Omron Sysmac Studio project Cobot Modbus Test_100221 (Sysmac Studio 1.40.0.64008, StandardProject)

# Controller new_Controller_0: NX102-9020 version 1.34
Units and slaves: Unit 1 : NX-OC4633 (N1)
Task PrimaryTask (priority 4, period or condition 2000): Main, TM_Movements_Connection, TM_Movements, CobotModbusComms
Library TM_Commands 1.2.1 (contents left out)
Library TMmodbus Lib FW1.80 FB3.0.03 3.0.03 (contents left out)

VAR_GLOBAL RETAIN
    StartCommunications : BOOL;  (* published *)
END_VAR
VAR_GLOBAL
    MBerror : WORD;  (* published *)
    RobotCoordinates : TMmodbus\sRobotCoordinate;  (* published *)
    TouchCoordinates : TMmodbus\sRobotCoordinateTouch;  (* published *)
    RobotStatus : TMmodbus\sRobotStatus;  (* published *)
    RobotVitals : TMmodbus\sRobotVitals;  (* published *)
    Config : TMmodbus\sConfiguration;  (* published *)
    RobotJointTorques : TMmodbus\sRobotJointTorque;  (* published *)
    RobotTCPLive : TMmodbus\sRobotTCPLive;  (* published *)
    CurrentProjectName : string[200];  (* published *)
    NewProjectName : string[200];  (* published *)
    CommsRoundRobin : REAL;  (* published *)
    TCPerror : WORD;  (* published *)
    RobotControlBoxInfo : TMmodbus\sRobotControllerData;  (* published *)
    Buttons : TMmodbus\sRobotStickButtons;  (* published *)
    RobotIO : TMmodbus\sRobotIO;  (* published *)
    RobotSafetySettings : TMmodbus\sRobotSafety;  (* published *)
    RealsToRobot : ARRAY[0..49] OF real;  (* published *)
    FloatsFromRobot : ARRAY[0..49] OF real;  (* published *)
    BoolsToRobot : ARRAY[0..63] OF BOOL;  (* published *)
    Int16sFromRobot : ARRAY[0..49] OF INT;  (* published *)
    BoolsFromRobot : ARRAY[0..63] OF BOOL;  (* published *)
    IntsToRobot : ARRAY[0..49] OF INT;  (* published *)
    CommunicationsStatus : _eCONNECTION_STATE;  (* published *)
    CommunicationsBusy : BOOL;  (* published *)
    TCPerrorOriginator : TMModbus\eFunctionBlockError;  (* published *)
    RetryCounter : UINT;  (* published *)
    Stitching_Status : DINT;  (* published *)
    Stitching_Speed : REAL;  (* published *)
    Robot_Status : DINT;  (* published *)
    RobPos_X : REAL;  (* published *)
    RobPos_Y : REAL;  (* published *)
    RobPos_Z : REAL;  (* published *)
    Relay_Output : BYTE;  (* at IOBus://unit#1/Output Bit 8 bits; published *)
    Relay_Output1 : BOOL;  (* at IOBus://unit#1/Output Bit 8 bits/Output Bit 00; published *)
    Relay_Output2 : BOOL;  (* at IOBus://unit#1/Output Bit 8 bits/Output Bit 01; published *)
    Relay_Output3 : BOOL;  (* at IOBus://unit#1/Output Bit 8 bits/Output Bit 02; published *)
    Relay_Output4 : BOOL;  (* at IOBus://unit#1/Output Bit 8 bits/Output Bit 03; published *)
    Run_Stiching : BOOL;  (* published *)
    StartProgram : BOOL;  (* published *)
    CableConnected : BOOL;  (* published *)
    MTCP_Connect_TCP_Socket : _sSOCKET;  (* published *)
    MTCP_Connect_Connected : BOOL;
    ListenNode_Connect_Connected : BOOL;
    ListenNode_Connect_TCP_Socket : _sSOCKET;
    TaskTimeFB : REAL;
    Speed : REAL;  (* published *)
    TM_ReadPosition_X : REAL;
    TM_ReadPosition_Y : REAL;
    TM_ReadPosition_Z : REAL;  (* published *)
    Register : ARRAY[0..1023] OF WORD;
    TM_MovCmd_Command : STRING[256];
    Stitching_InManual : BOOL;
    Vision_IN : ARRAY[0..495] OF BYTE;  (* network input *)
    Vision_IN_Bit : ARRAY[0..11] OF BYTE;  (* network input *)
    Vision_Out_Bit : ARRAY[0..11] OF BYTE;  (* network output *)
    Vision_OUT : ARRAY[0..495] OF BYTE;  (* network output *)
END_VAR

PROGRAM Main
VAR
    Input1 : BOOL;  (* Enter Variable Commen *)
    Input2 : BOOL;
    Input3 : BOOL;
    Input4 : BOOL;
    RobotPos_Stiching : BOOL;
    xPlaceholder : DINT;
    yPlaceholder : DINT;
    zPlaceholder : DINT;
    placeholder : BOOL;
    Robot_Running : BOOL;
    Rb_Error_Present : BOOL;
    St_Error_Present : BOOL;
    CommunicationsBusy : BOOL;
    StartCommunications : BOOL;
    Start : BOOL;
    test : BOOL;
    def : BOOL;
    Angle : BOOL;
    Part_Orientation : INT;
    Part_Orientation_REAL : REAL;
    Part_Orientation_DINT : DINT;
    Part_Dist_X : DINT;
    Part_Dist_Y : DINT;
END_VAR
VAR_EXTERNAL
    Stitching_Status : DINT;
    Stitching_Speed : REAL;
    Robot_Status : DINT;
    Relay_Output : BYTE;
    RobPos_X : REAL;
    RobPos_Y : REAL;
    RobPos_Z : REAL;
    RobotCoordinates : TMmodbus\sRobotCoordinate;
    RobotStatus : TMmodbus\sRobotStatus;
    Run_Stiching : BOOL;
    Speed : REAL;
    Vision_IN : ARRAY[0..495] OF BYTE;
END_VAR

(* Section DataToGrafana: ladder, written here as Structured Text *)

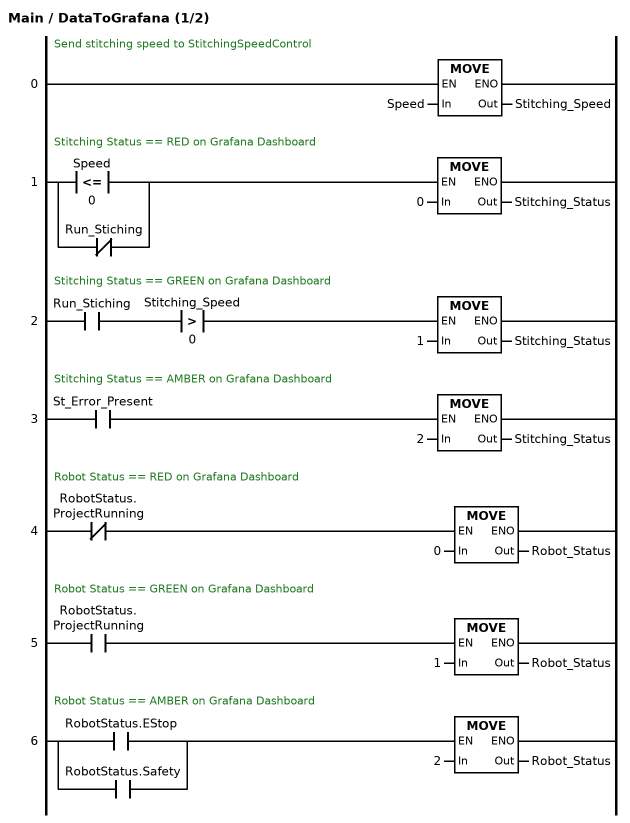
(* Rung 0: Send stitching speed to StitchingSpeedControl *)
Stitching_Speed := Speed;
(* Rung 1: Stitching Status == RED on Grafana Dashboard *)
IF (Speed <= 0) OR NOT Run_Stiching THEN Stitching_Status := 0; END_IF;
(* Rung 2: Stitching Status == GREEN on Grafana Dashboard *)
IF Run_Stiching AND (Stitching_Speed > 0) THEN Stitching_Status := 1; END_IF;
(* Rung 3: Stitching Status == AMBER on Grafana Dashboard *)
IF St_Error_Present THEN Stitching_Status := 2; END_IF;
(* Rung 4: Robot Status == RED on Grafana Dashboard *)
IF NOT RobotStatus.ProjectRunning THEN Robot_Status := 0; END_IF;
(* Rung 5: Robot Status == GREEN on Grafana Dashboard *)
IF RobotStatus.ProjectRunning THEN Robot_Status := 1; END_IF;
(* Rung 6: Robot Status == AMBER on Grafana Dashboard *)
IF RobotStatus.EStop OR RobotStatus.Safety THEN Robot_Status := 2; END_IF;

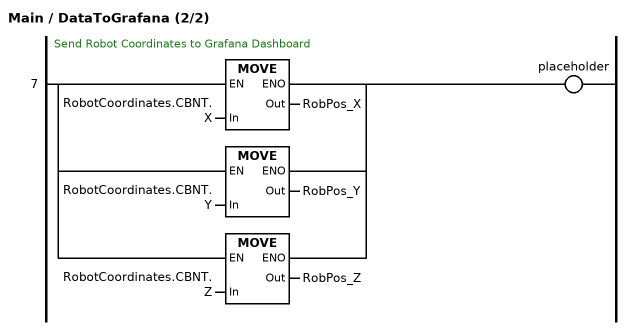
(* Rung 7: Send Robot Coordinates to Grafana Dashboard *)
RobPos_X := RobotCoordinates.CBNT.X;
RobPos_Y := RobotCoordinates.CBNT.Y;
RobPos_Z := RobotCoordinates.CBNT.Z;
placeholder := TRUE;

(* Section StichingSpeedControl: ladder, written here as Structured Text *)

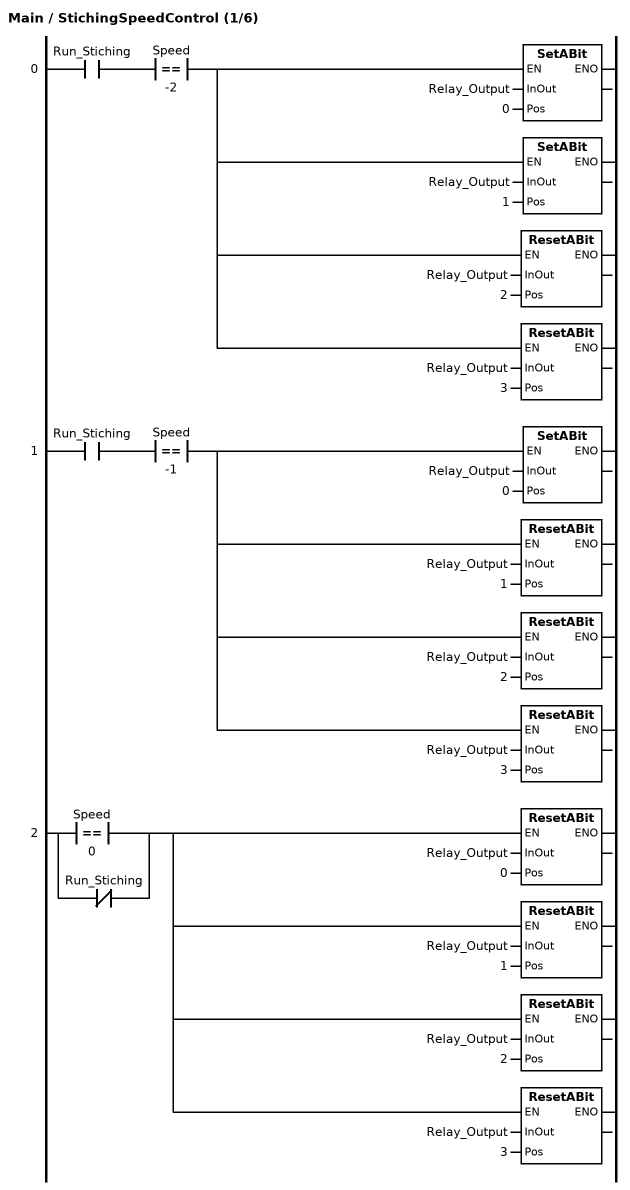
(* Rung 0 *)
IF Run_Stiching AND (Speed = -2) THEN
    SetABit(InOut := Relay_Output, Pos := 0);
    SetABit(InOut := Relay_Output, Pos := 1);
    ResetABit(InOut := Relay_Output, Pos := 2);
    ResetABit(InOut := Relay_Output, Pos := 3);
END_IF;
(* Rung 1 *)
IF Run_Stiching AND (Speed = -1) THEN
    SetABit(InOut := Relay_Output, Pos := 0);
    ResetABit(InOut := Relay_Output, Pos := 1);
    ResetABit(InOut := Relay_Output, Pos := 2);
    ResetABit(InOut := Relay_Output, Pos := 3);
END_IF;
(* Rung 2 *)
IF (Speed = 0) OR NOT Run_Stiching THEN
    ResetABit(InOut := Relay_Output, Pos := 0);
    ResetABit(InOut := Relay_Output, Pos := 1);
    ResetABit(InOut := Relay_Output, Pos := 2);
    ResetABit(InOut := Relay_Output, Pos := 3);
END_IF;

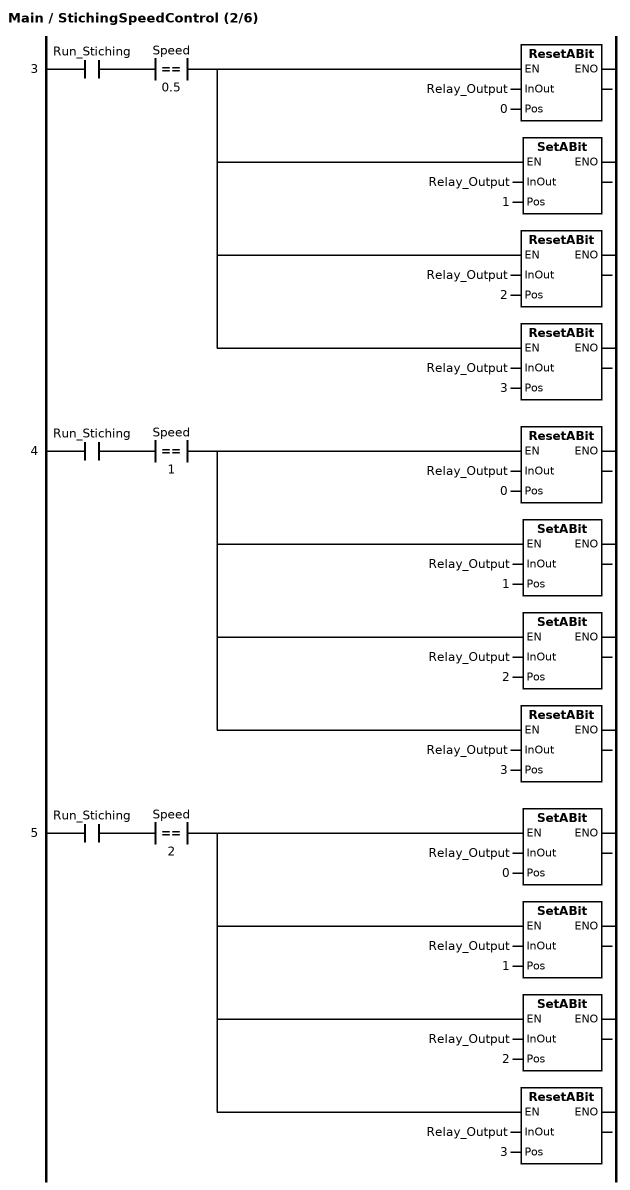
(* Rung 3 *)
IF Run_Stiching AND (Speed = 0.5) THEN
    ResetABit(InOut := Relay_Output, Pos := 0);
    SetABit(InOut := Relay_Output, Pos := 1);
    ResetABit(InOut := Relay_Output, Pos := 2);
    ResetABit(InOut := Relay_Output, Pos := 3);
END_IF;
(* Rung 4 *)
IF Run_Stiching AND (Speed = 1) THEN
    ResetABit(InOut := Relay_Output, Pos := 0);
    SetABit(InOut := Relay_Output, Pos := 1);
    SetABit(InOut := Relay_Output, Pos := 2);
    ResetABit(InOut := Relay_Output, Pos := 3);
END_IF;
(* Rung 5 *)
IF Run_Stiching AND (Speed = 2) THEN
    SetABit(InOut := Relay_Output, Pos := 0);
    SetABit(InOut := Relay_Output, Pos := 1);
    SetABit(InOut := Relay_Output, Pos := 2);
    ResetABit(InOut := Relay_Output, Pos := 3);
END_IF;

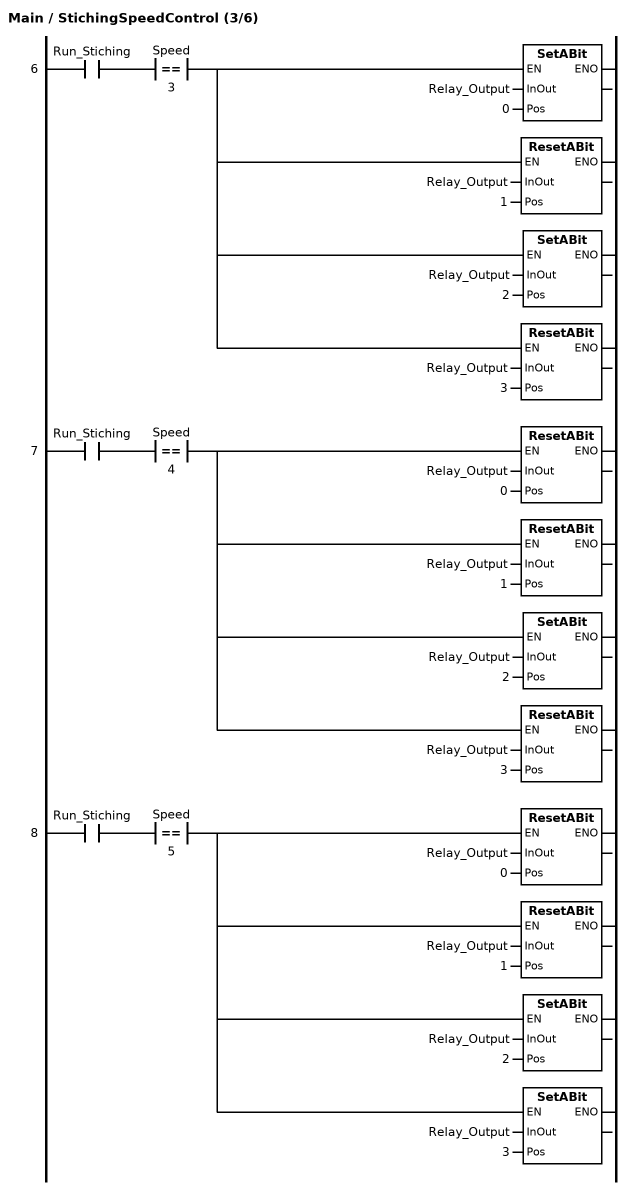
(* Rung 6 *)
IF Run_Stiching AND (Speed = 3) THEN
    SetABit(InOut := Relay_Output, Pos := 0);
    ResetABit(InOut := Relay_Output, Pos := 1);
    SetABit(InOut := Relay_Output, Pos := 2);
    ResetABit(InOut := Relay_Output, Pos := 3);
END_IF;
(* Rung 7 *)
IF Run_Stiching AND (Speed = 4) THEN
    ResetABit(InOut := Relay_Output, Pos := 0);
    ResetABit(InOut := Relay_Output, Pos := 1);
    SetABit(InOut := Relay_Output, Pos := 2);
    ResetABit(InOut := Relay_Output, Pos := 3);
END_IF;
(* Rung 8 *)
IF Run_Stiching AND (Speed = 5) THEN
    ResetABit(InOut := Relay_Output, Pos := 0);
    ResetABit(InOut := Relay_Output, Pos := 1);
    SetABit(InOut := Relay_Output, Pos := 2);
    SetABit(InOut := Relay_Output, Pos := 3);
END_IF;

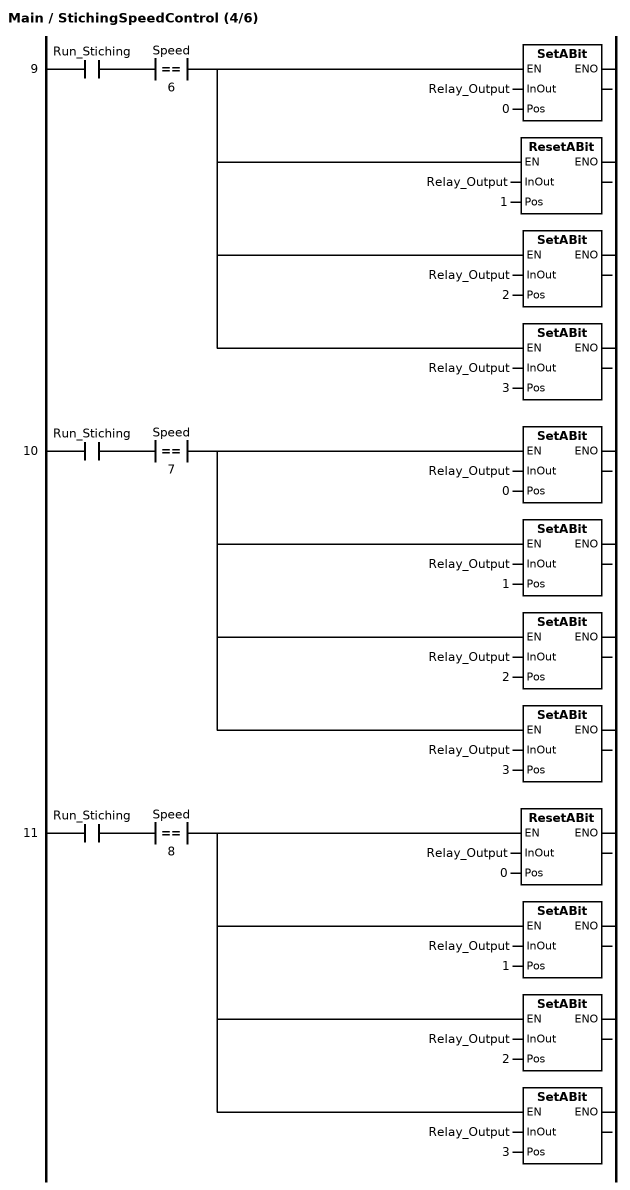
(* Rung 9 *)
IF Run_Stiching AND (Speed = 6) THEN
    SetABit(InOut := Relay_Output, Pos := 0);
    ResetABit(InOut := Relay_Output, Pos := 1);
    SetABit(InOut := Relay_Output, Pos := 2);
    SetABit(InOut := Relay_Output, Pos := 3);
END_IF;
(* Rung 10 *)
IF Run_Stiching AND (Speed = 7) THEN
    SetABit(InOut := Relay_Output, Pos := 0);
    SetABit(InOut := Relay_Output, Pos := 1);
    SetABit(InOut := Relay_Output, Pos := 2);
    SetABit(InOut := Relay_Output, Pos := 3);
END_IF;
(* Rung 11 *)
IF Run_Stiching AND (Speed = 8) THEN
    ResetABit(InOut := Relay_Output, Pos := 0);
    SetABit(InOut := Relay_Output, Pos := 1);
    SetABit(InOut := Relay_Output, Pos := 2);
    SetABit(InOut := Relay_Output, Pos := 3);
END_IF;

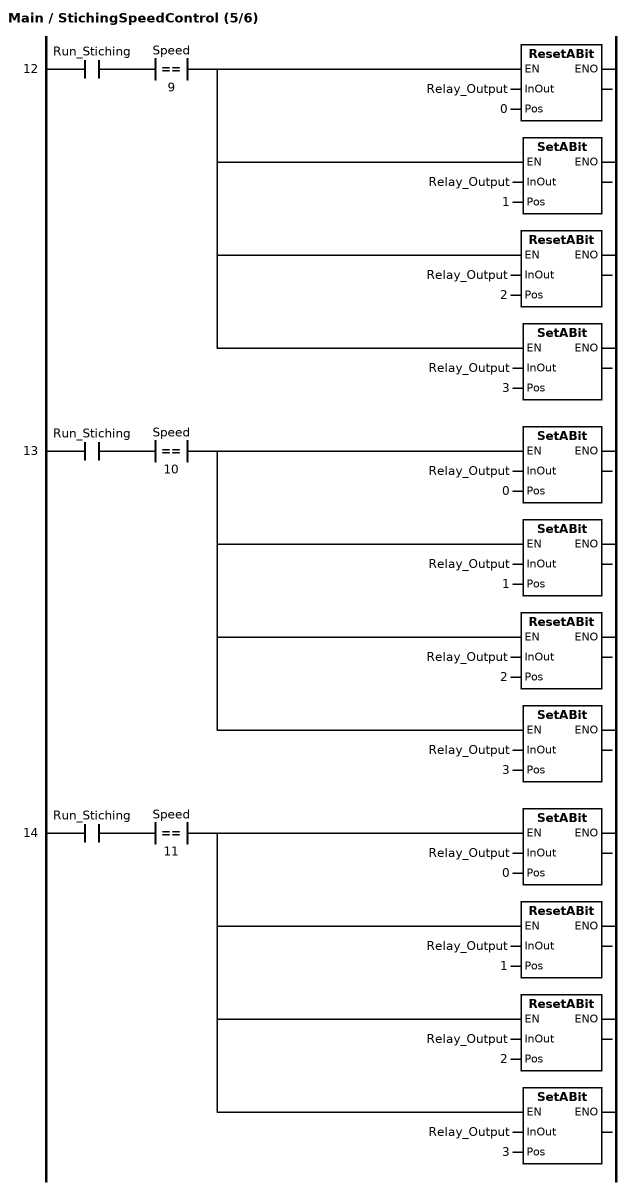
(* Rung 12 *)
IF Run_Stiching AND (Speed = 9) THEN
    ResetABit(InOut := Relay_Output, Pos := 0);
    SetABit(InOut := Relay_Output, Pos := 1);
    ResetABit(InOut := Relay_Output, Pos := 2);
    SetABit(InOut := Relay_Output, Pos := 3);
END_IF;
(* Rung 13 *)
IF Run_Stiching AND (Speed = 10) THEN
    SetABit(InOut := Relay_Output, Pos := 0);
    SetABit(InOut := Relay_Output, Pos := 1);
    ResetABit(InOut := Relay_Output, Pos := 2);
    SetABit(InOut := Relay_Output, Pos := 3);
END_IF;
(* Rung 14 *)
IF Run_Stiching AND (Speed = 11) THEN
    SetABit(InOut := Relay_Output, Pos := 0);
    ResetABit(InOut := Relay_Output, Pos := 1);
    ResetABit(InOut := Relay_Output, Pos := 2);
    SetABit(InOut := Relay_Output, Pos := 3);
END_IF;

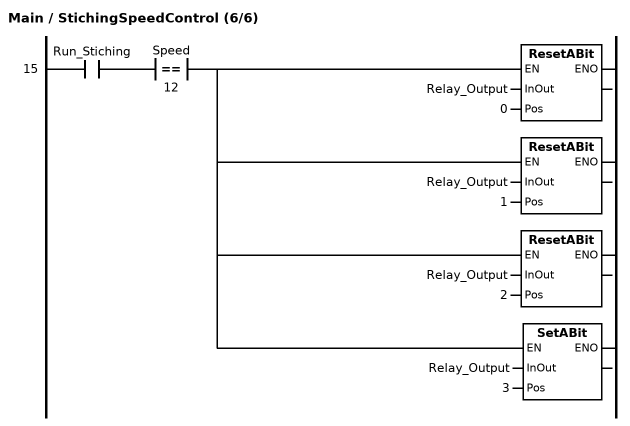
(* Rung 15 *)
IF Run_Stiching AND (Speed = 12) THEN
    ResetABit(InOut := Relay_Output, Pos := 0);
    ResetABit(InOut := Relay_Output, Pos := 1);
    ResetABit(InOut := Relay_Output, Pos := 2);
    SetABit(InOut := Relay_Output, Pos := 3);
END_IF;

(* Section VisionComms: ladder, written here as Structured Text *)

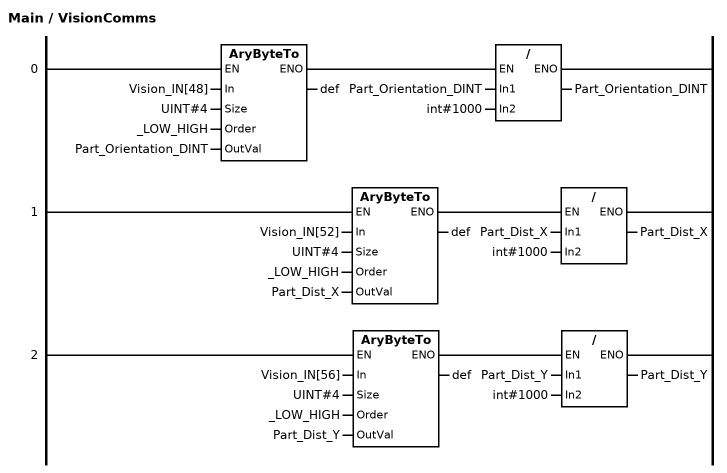
(* Rung 0 *)
def := AryByteTo(In := Vision_IN[48], Size := UINT#4, Order := _LOW_HIGH, OutVal := Part_Orientation_DINT);
Part_Orientation_DINT := Part_Orientation_DINT / int#1000;
(* Rung 1 *)
def := AryByteTo(In := Vision_IN[52], Size := UINT#4, Order := _LOW_HIGH, OutVal := Part_Dist_X);
Part_Dist_X := Part_Dist_X / int#1000;
(* Rung 2 *)
def := AryByteTo(In := Vision_IN[56], Size := UINT#4, Order := _LOW_HIGH, OutVal := Part_Dist_Y);
Part_Dist_Y := Part_Dist_Y / int#1000;
END_PROGRAM

PROGRAM TM_Movements_Connection
VAR
    ListenNode_Connect_Instance : ListenNode_Connect;
    ListenNode_Connect_Enable : BOOL;
    ListenNode_Connect_IPaddress : STRING[16];
    ListenNode_Connect_Port : UINT;
    ListenNode_Connect_Connect : BOOL;
    ListenNode_Connect_Error : BOOL;
    ListenNode_Connect_ErrorID : WORD;
    ListenNode_Connect_EtnConnError : BOOL;
    ListenNode_Connect_Socket_Status : _eCONNECTION_STATE;
END_VAR
VAR_EXTERNAL
    ListenNode_Connect_Connected : BOOL;
    ListenNode_Connect_TCP_Socket : _sSOCKET;
    StartProgram : BOOL;
END_VAR
ListenNode_Connect_Enable:=TRUE;
ListenNode_Connect_IPaddress:='10.1.20.60';
ListenNode_Connect_Port:=5890;

ListenNode_Connect_Connect:=StartProgram;

ListenNode_Connect_Instance(
	Enable:=ListenNode_Connect_Enable,
	IPaddress:=ListenNode_Connect_IPaddress,
	Port:=ListenNode_Connect_Port,
	Connect:=ListenNode_Connect_Connect,
	Connected=>ListenNode_Connect_Connected,
	Error=>ListenNode_Connect_Error,
	ErrorID=>ListenNode_Connect_ErrorID,
	EtnConnError=>ListenNode_Connect_EtnConnError,
	TCP_Socket=>ListenNode_Connect_TCP_Socket,
	Socket_Status=>ListenNode_Connect_Socket_Status
);
END_PROGRAM

PROGRAM TM_Movements
VAR
    TM_ChangeLoad_Instance : TM_ChangeLoad;
    TM_ChangeTCP_Instance : TM_ChangeTCP;
    TM_MovCmd_Instance : TM_MovCmd;
    TM_MovCmd_Done : BOOL;
    TM_MovCmd_Busy : BOOL;
    TM_MovCmd_Error : BOOL;
    TM_MovCmd_ErrorID : WORD;
    TM_MovCmd_Execute : BOOL;
    TM_MovCmd_Movement : STRING[256];
    TM_MovCmd_DataFormat : STRING[256];
    DD_ListenNode_Connect_Connected : F_TRIG;
    TM_MovCmd_Point : STRING[256];
    TM_MovCmd_Speed : INT;
    TM_MovCmd_AccelTime : INT;
    TM_MovCmd_Blending : INT;
    TM_MovCmd_PrecisePos : BOOL;
    TM_MovCmd_RobotPose : STRING[256];
    TM_MovCmd_ActivateExit : BOOL;
    TM_MovCmd_CommandID : INT;
    Enable : BOOL;
    DU_Enable : R_TRIG;
    TM_ChangeBase_Busy : BOOL;
    TM_ChangeBase_Done : BOOL;
    TM_ChangeBase_Error : BOOL;
    TM_ChangeBase_ErrorID : WORD;
    TM_ChangeBase_Execute : BOOL;
    TM_ChangeBase_Base : STRING[256];
    TM_ChangeBase_ActivateExit : BOOL;
    TM_ChangeBase_CommandID : INT;
    TM_ChangeLoad_Execute : BOOL;
    TM_ChangeLoad_Busy : BOOL;
    TM_ChangeLoad_Done : BOOL;
    TM_ChangeLoad_Error : BOOL;
    TM_ChangeLoad_ErrorID : WORD;
    TM_ChangeLoad_Payload : STRING[256];
    TM_ChangeLoad_ActivateExit : BOOL;
    TM_ChangeLoad_CommandID : INT;
    TM_ChangeTCP_Busy : BOOL;
    TM_ChangeTCP_Done : BOOL;
    TM_ChangeTCP_Error : BOOL;
    TM_ChangeTCP_ErrorID : WORD;
    TM_ChangeTCP_Execute : BOOL;
    TM_ChangeTCP_TCP : STRING[256];
    TM_ChangeTCP_Weight : STRING[256];
    TM_ChangeTCP_MomInertia : STRING[256];
    TM_ChangeTCP_RefFrame : STRING[256];
    TM_ChangeTCP_ActivateExit : BOOL;
    TM_ChangeTCP_CommandID : INT;
    TM_CircleCmd_Done : BOOL;
    TM_CircleCmd_Busy : BOOL;
    TM_CircleCmd_Error : BOOL;
    TM_CircleCmd_ErrorID : WORD;
    TM_CircleCmd_Execute : BOOL;
    TM_CircleCmd_DataFormat : STRING[256];
    TM_CircleCmd_ArcPoint : STRING[256];
    TM_CircleCmd_EndArcPoint : STRING[256];
    TM_CircleCmd_Speed : INT;
    TM_CircleCmd_AccelTime : INT;
    TM_CircleCmd_Blending : INT;
    TM_CircleCmd_ArcAngle : INT;
    TM_CircleCmd_PrecisePos : BOOL;
    TM_CircleCmd_Command : STRING[256];
    TM_CircleCmd_ActivateExit : BOOL;
    TM_CircleCmd_CommandID : INT;
    PickPoint : STRING[256];
    PalletFirstPoint : STRING[256];
    StartPoint : STRING[256];
    PalletSecondPoint : STRING[256];
    PalletThirdPoint : STRING[256];
    PalletFourthPoint : STRING[256];
    MovementIndicatorStage : INT;
    DownRelative : STRING[256];
    HighRelative : STRING[256];
    TM_ChangeBase_Command : STRING[256];
    TM_ChangeLoad_Command : STRING[256];
    TM_ChangeTCP_Command : STRING[256];
    DD_CableConnected : F_TRIG;
    TM_MovCmd_ListenNode : STRING[256];
    Stage : INT;
    TM_MovCmd_TimeOutET : TIME;
    TM_MovCmd_Enable : BOOL;
    TM_ChangeTCP_Enable : BOOL;
    TM_ChangeTCP_ListenNode : STRING[256];
    TM_ChangeTCP_TimeOutET : TIME;
    TM_ChangeLoad_Enable : BOOL;
    TM_ChangeLoad_ListenNode : STRING[256];
    TM_ChangeLoad_TimeOutET : TIME;
    TM_CircleCmd_Instance : TM_CircleCmd;
    TM_ChangeBase_Instance : TM_ChangeBase;
    TM_ChangeBase_Enable : BOOL;
    TM_CircleCmd_Enable : BOOL;
    TM_CircleCmd_ListenNode : STRING[256];
    TM_CircleCmd_TimeOutET : TIME;
    TM_ChangeBase_ListenNode : STRING[256];
    TM_ChangeBase_TimeOutET : TIME;
    Home : STRING[256];
    Midpoint : STRING[256];
    Approach : STRING[256];
    Attach : STRING[256];
    Position1 : STRING[256];
    Position3 : STRING[256];
    Position2 : STRING[256];
    Position4 : STRING[256];
    Position5 : STRING[256];
    Position6 : STRING[256];
    Position7 : STRING[256];
    Position8 : STRING[256];
    Position9 : STRING[256];
    Position10 : STRING[256];
    Position11 : STRING[256];
END_VAR
VAR_EXTERNAL
    StartProgram : BOOL;
    CableConnected : BOOL;
    ListenNode_Connect_Connected : BOOL;
    ListenNode_Connect_TCP_Socket : _sSOCKET;
    Run_Stiching : BOOL;
    Stitching_Speed : REAL;
    Speed : REAL;
    TM_ReadPosition_X : REAL;
    TM_ReadPosition_Y : REAL;
    TM_ReadPosition_Z : REAL;
    TM_MovCmd_Command : STRING[256];
    RobPos_X : REAL;
    RobotIO : TMmodbus\sRobotIO;
    Stitching_InManual : BOOL;
END_VAR
DU_Enable(Clk:=Enable);
DD_ListenNode_Connect_Connected(Clk:=ListenNode_Connect_Connected);
DD_CableConnected(Clk:=CableConnected);

Enable:=StartProgram;

IF DU_Enable.Q THEN
	
	Stage:=0;
	MovementIndicatorStage:=0;
	
	//Robot points in the format 'X,Y,Z,Rx,Ry,Rz)
	Home:= '295.985,-353.326,669.109,-178.747,1.530,-175.599';
	Midpoint:='329.186,-372.735,470.938,-179.247,0.828,-175.618';
	Approach:='338.482,-378.188,292.444,-179.411,0.606,-175.625';
	Attach:='340.242,-379.659,136.197,-179.411,0.606,-175.625';
	Position1:='532.31,-376.88,141.62,-179.10,0.61,-168.20';
	Position2:='644.42,-183.83,140.96,-179.14,0.66,-171.77';
	Position3:='764.70,42.23,139.59,-179.14,.066,-171.77';
	Position4:='761.007,78.442,138.293,-179.146,-0.090,-169.031';
	 //Start of Stitching
	Position5:='772.437,138.944,139.413,-179.670,1.537,-178.155';
	Position6:='812.470,204.177,142.787,178.907,5.421,-175.081';
	Position7:='876.098,332.162,135.333,176.349,12.256,-169.988';
	Position8:='893.624,371.169,139.251,178.969,5.285,-168.090';
	Position9:='898.806,414.795,127.072,179.563,3.650,-166.038';
	Position10:='292.268,-351.946,693.455,-179.506,-0.892,-179.089';
	
	
END_IF;

IF DD_ListenNode_Connect_Connected.Q OR DD_CableConnected.Q THEN //connection closed or cable disconnected.
	
	Stage:= 9999; //MovementIndicatorStage;
	
END_IF;

IF Enable AND ListenNode_Connect_Connected AND CableConnected THEN	//the PLC program is enabled and there is connection with listen node and the cable is connected
	
	CASE Stage OF
		
		//-----------------------------------------------------------TCP Selection--------------------------------------------------
		0:
			TM_ChangeTCP_Enable:=FALSE;
			IF (NOT TM_ChangeTCP_Done) AND (NOT TM_ChangeTCP_Error) AND (NOT TM_ChangeTCP_Busy) THEN
				Stage:=1; 
			END_IF;
		1:
			TM_ChangeTCP_Enable:=TRUE;	
			TM_ChangeTCP_ActivateExit:=TRUE;
			TM_ChangeTCP_CommandID:=1;
			TM_ChangeTCP_Execute:=FALSE;
			TM_ChangeTCP_ListenNode:='Listen1';
			TM_ChangeTCP_TCP:='TestTool';
			TM_MovCmd_Command:='var_Start_Stitching=10';
			TM_ChangeTCP_Weight:='';
			TM_ChangeTCP_MomInertia:='';
			TM_ChangeTCP_RefFrame:='';
			TM_ChangeLoad_Payload:='';
			IF (NOT TM_ChangeTCP_Done) AND (NOT TM_ChangeTCP_Error) THEN
				Stage:=2;
			END_IF;
		2:
			TM_ChangeTCP_Execute:=TRUE;
			IF TM_ChangeTCP_Done THEN
				Stage:=10;
			ELSIF TM_ChangeTCP_Error THEN
				Stage:=9999;
			END_IF;
		//-----------------------------------------------------------Program Stages--------------------------------------------------------------
		10:
			TM_MovCmd_Enable:=FALSE;
			MovementIndicatorStage:=Stage;
			IF (NOT TM_MovCmd_Done) AND (NOT TM_MovCmd_Error) AND (NOT TM_MovCmd_Busy) THEN
				Stage:=11;
			END_IF;
		11:
			TM_MovCmd_Enable:=TRUE;
			TM_MovCmd_Movement:='PTP';
			TM_MovCmd_DataFormat:='CPP';
			TM_MovCmd_Point:=Home;
			TM_MovCmd_Speed:=50;
			TM_MovCmd_AccelTime:=200;
			TM_MovCmd_Blending:=100;
			TM_MovCmd_PrecisePos:=1;
			TM_MovCmd_RobotPose:='';
			TM_MovCmd_Command:='var_Start_Stitching=10';
			TM_MovCmd_ActivateExit:=TRUE;
			TM_MovCmd_CommandID:=1;
			TM_MovCmd_Execute:=FALSE;
			TM_MovCmd_ListenNode:='Listen1';
			IF (NOT TM_MovCmd_Done) AND (NOT TM_MovCmd_Error) THEN
				Stage:=12;
			END_IF;
		12:
			TM_MovCmd_Execute:=TRUE;
			IF TM_MovCmd_Done THEN
				Stage:=20;
			ELSIF TM_MovCmd_Error THEN
				Stage:=9999;
			END_IF;
		20:
			TM_MovCmd_Enable:=FALSE;
			MovementIndicatorStage:=Stage;
			IF (NOT TM_MovCmd_Done) AND (NOT TM_MovCmd_Error) AND (NOT TM_MovCmd_Busy) THEN
				Stage:=31;
			END_IF;
		21:			
			TM_MovCmd_Enable:=TRUE;
			TM_MovCmd_Movement:='PTP';
			TM_MovCmd_DataFormat:='CPP';
			TM_MovCmd_Point:=Midpoint;
			TM_MovCmd_Speed:=50;
			TM_MovCmd_AccelTime:=200;
			TM_MovCmd_Blending:=100;
			TM_MovCmd_PrecisePos:=1;
			TM_MovCmd_RobotPose:='';
			TM_MovCmd_Command:='var_Start_Stitching=10';
			TM_MovCmd_ActivateExit:=FALSE;
			TM_MovCmd_CommandID:=1;
			TM_MovCmd_Execute:=FALSE;
			TM_MovCmd_ListenNode:='Listen1';
			IF (NOT TM_MovCmd_Done) AND (NOT TM_MovCmd_Error) THEN
				Stage:=22;
			END_IF;			
		22:
			TM_MovCmd_Execute:=TRUE;
			IF TM_MovCmd_Done THEN
				Stage:=30;
			ELSIF TM_MovCmd_Error THEN
				Stage:=9999;
			END_IF;
		30:
			TM_MovCmd_Enable:=FALSE;
			IF (NOT TM_MovCmd_Done) AND (NOT TM_MovCmd_Error) AND (NOT TM_MovCmd_Busy) THEN
				Stage:=31;
			END_IF;
		31:			
			TM_MovCmd_Enable:=TRUE;
			TM_MovCmd_Movement:='PTP';
			TM_MovCmd_DataFormat:='CPP';
			TM_MovCmd_Point:=Approach;
			TM_MovCmd_Speed:=50;
			TM_MovCmd_AccelTime:=200;
			TM_MovCmd_Blending:=100;
			TM_MovCmd_PrecisePos:=1;
			TM_MovCmd_RobotPose:='';
			TM_MovCmd_Command:='var_Start_Stitching=10';
			TM_MovCmd_ActivateExit:=FALSE;
			TM_MovCmd_CommandID:=1;
			TM_MovCmd_Execute:=FALSE;
			TM_MovCmd_ListenNode:='Listen1';
			IF (NOT TM_MovCmd_Done) AND (NOT TM_MovCmd_Error) THEN
				Stage:=32;
			END_IF;
		
		32:
			TM_MovCmd_Execute:=TRUE;
			IF TM_MovCmd_Done THEN
				Stage:=50;
			ELSIF TM_MovCmd_Error THEN
				Stage:=9999;
			END_IF;
		//////////////////////////////////////////////////////////////////////////////////////////////
		//Not used at the moment
		40:
			TM_ChangeLoad_Enable:=FALSE;
			IF (NOT TM_ChangeLoad_Done) AND (NOT TM_ChangeLoad_Error) AND (NOT TM_ChangeLoad_Busy) THEN
				Stage:=41;
			END_IF;
		41:
			TM_ChangeLoad_Enable:=TRUE;	 
			TM_ChangeLoad_ActivateExit:=TRUE;
			TM_ChangeLoad_CommandID:=1;
			TM_ChangeLoad_Execute:=FALSE;
			TM_ChangeLoad_ListenNode:='Listen1';
			TM_ChangeLoad_Payload:='0.1';
			IF (NOT TM_ChangeLoad_Done) AND (NOT TM_ChangeLoad_Error) THEN
				Stage:=42;
			END_IF;
		42:
			TM_ChangeLoad_Execute:=TRUE;
			IF TM_ChangeLoad_Done THEN
				Stage:=50;
			ELSIF TM_ChangeLoad_Error THEN
				Stage:=9999;
			END_IF;			
		//////////////////////////////////////////////////////////////////////////////////	
		50:
			TM_MovCmd_Enable:=FALSE;
			IF (NOT TM_MovCmd_Done) AND (NOT TM_MovCmd_Error) AND (NOT TM_MovCmd_Busy) THEN
				Stage:=51;
			END_IF;	
		51:
			TM_MovCmd_Enable:=TRUE;
			TM_MovCmd_Movement:='Line';
			TM_MovCmd_DataFormat:='CPR';
			TM_MovCmd_Point:=Attach;
			TM_MovCmd_Speed:=50;
			TM_MovCmd_AccelTime:=200;
			TM_MovCmd_Blending:=100;
			TM_MovCmd_PrecisePos:=1;
			TM_MovCmd_RobotPose:='';
			TM_MovCmd_Command:='var_Start_Stitching=10';
			TM_MovCmd_ActivateExit:=FALSE;
			TM_MovCmd_CommandID:=1;
			TM_MovCmd_Execute:=FALSE;
			TM_MovCmd_ListenNode:='Listen1';
			IF (NOT TM_MovCmd_Done) AND (NOT TM_MovCmd_Error) THEN
				Stage:=52;
			END_IF;
		52:
			TM_MovCmd_Execute:=TRUE;
			IF TM_MovCmd_Done THEN
				Stage:=70;
			ELSIF TM_MovCmd_Error THEN
				Stage:=9999;
			END_IF;
		60:
			TM_MovCmd_Enable:=FALSE;
			MovementIndicatorStage:=Stage;
			IF (NOT TM_MovCmd_Done) AND (NOT TM_MovCmd_Error) AND (NOT TM_MovCmd_Busy) THEN
				Stage:=61;
			END_IF;	
		
		61:
			TM_MovCmd_Enable:=TRUE;
			TM_MovCmd_Movement:='Line';
			TM_MovCmd_DataFormat:='CPR';
			TM_MovCmd_Point:=Approach;
			TM_MovCmd_Speed:=50;
			TM_MovCmd_AccelTime:=200;
			TM_MovCmd_Blending:=100;
			TM_MovCmd_PrecisePos:=1;
			TM_MovCmd_RobotPose:='';
			TM_MovCmd_Command:='var_Start_Stitching=10';
			TM_MovCmd_ActivateExit:=FALSE;
			TM_MovCmd_CommandID:=1;
			TM_MovCmd_Execute:=FALSE;
			TM_MovCmd_ListenNode:='Listen1';
			IF (NOT TM_MovCmd_Done) AND (NOT TM_MovCmd_Error) THEN
				Stage:=62;
			END_IF;
		62:
			TM_MovCmd_Execute:=TRUE;
			IF TM_MovCmd_Done THEN
				Stage:=70;
			ELSIF TM_MovCmd_Error THEN
				Stage:=9999;
			END_IF;
			
		70:
			TM_MovCmd_Enable:=FALSE;
			MovementIndicatorStage:=Stage;
			IF (NOT TM_MovCmd_Done) AND (NOT TM_MovCmd_Error) AND (NOT TM_MovCmd_Busy) THEN
				Stage:=71;
			END_IF;	
		
		71:
			TM_MovCmd_Enable:=TRUE;
			TM_MovCmd_Movement:='Line';
			TM_MovCmd_DataFormat:='CPR';
			TM_MovCmd_Point:=Position1;
			TM_MovCmd_Speed:=50;
			TM_MovCmd_AccelTime:=200;
			TM_MovCmd_Blending:=100;
			TM_MovCmd_PrecisePos:=0;
			TM_MovCmd_RobotPose:='';
			TM_MovCmd_Command:='var_Start_Stitching=10';
			TM_MovCmd_ActivateExit:=FALSE;
			TM_MovCmd_CommandID:=1;
			TM_MovCmd_Execute:=FALSE;
			TM_MovCmd_ListenNode:='Listen1';
			IF (NOT TM_MovCmd_Done) AND (NOT TM_MovCmd_Error) THEN
				Stage:=72;
			END_IF;
		72:
			TM_MovCmd_Execute:=TRUE;
			IF TM_MovCmd_Done THEN
				Stage:=80;
			ELSIF TM_MovCmd_Error THEN
				Stage:=9999;
			END_IF;
		80:
			TM_MovCmd_Enable:=FALSE;
			MovementIndicatorStage:=Stage;
			IF (NOT TM_MovCmd_Done) AND (NOT TM_MovCmd_Error) AND (NOT TM_MovCmd_Busy) THEN
				Stage:=81;
			END_IF;	
		
		81:
			TM_MovCmd_Enable:=TRUE;
			TM_MovCmd_Movement:='Line';
			TM_MovCmd_DataFormat:='CPR';
			TM_MovCmd_Point:=Position2;
			TM_MovCmd_Speed:=50;
			TM_MovCmd_AccelTime:=200;
			TM_MovCmd_Blending:=100;
			TM_MovCmd_PrecisePos:=0;
			TM_MovCmd_RobotPose:='';
			TM_MovCmd_Command:='var_Start_Stitching=10';
			TM_MovCmd_ActivateExit:=FALSE;
			TM_MovCmd_CommandID:=1;
			TM_MovCmd_Execute:=FALSE;
			TM_MovCmd_ListenNode:='Listen1';
			IF (NOT TM_MovCmd_Done) AND (NOT TM_MovCmd_Error) THEN
				Stage:=82;
			END_IF;
		82:
			TM_MovCmd_Execute:=TRUE;
			IF TM_MovCmd_Done THEN
				Stage:=90;
			ELSIF TM_MovCmd_Error THEN
				Stage:=9999;
			END_IF;
		90:
			TM_MovCmd_Enable:=FALSE;
			MovementIndicatorStage:=Stage;
			IF (NOT TM_MovCmd_Done) AND (NOT TM_MovCmd_Error) AND (NOT TM_MovCmd_Busy) THEN
				Stage:=91;
			END_IF;	
		
		91:
			TM_MovCmd_Enable:=TRUE;
			TM_MovCmd_Movement:='Line';
			TM_MovCmd_DataFormat:='CPR';
			TM_MovCmd_Point:=Position3;
			TM_MovCmd_Speed:=50;
			TM_MovCmd_AccelTime:=200;
			TM_MovCmd_Blending:=100;
			TM_MovCmd_PrecisePos:=1;
			TM_MovCmd_RobotPose:='';
			TM_MovCmd_Command:='var_Start_Stitching=10';
			TM_MovCmd_ActivateExit:=FALSE;
			TM_MovCmd_CommandID:=1;
			TM_MovCmd_Execute:=FALSE;
			TM_MovCmd_ListenNode:='Listen1';
		
			IF (NOT TM_MovCmd_Done) AND (NOT TM_MovCmd_Error) THEN
				Stage:=92;
			END_IF;
		92:
			TM_MovCmd_Execute:=TRUE;
			IF TM_MovCmd_Done THEN;
				Stage:=100;
			ELSIF TM_MovCmd_Error THEN
				Stage:=9999;
			END_IF;	
			
			100:
			TM_MovCmd_Enable:=FALSE;
			MovementIndicatorStage:=Stage;
			IF (NOT TM_MovCmd_Done) AND (NOT TM_MovCmd_Error) AND (NOT TM_MovCmd_Busy) THEN
				Stage:=101;
			END_IF;	
		
		101:
			TM_MovCmd_Enable:=TRUE;
			TM_MovCmd_Movement:='Line';
			TM_MovCmd_DataFormat:='CPR';
			TM_MovCmd_Point:=Position4;
			TM_MovCmd_Speed:=50;
			TM_MovCmd_AccelTime:=200;
			TM_MovCmd_Blending:=100;
			TM_MovCmd_PrecisePos:=1;
			TM_MovCmd_RobotPose:='';
			TM_MovCmd_Command:='var_Start_Stitching=10';
			TM_MovCmd_ActivateExit:=FALSE;
			TM_MovCmd_CommandID:=1;
			TM_MovCmd_Execute:=FALSE;
			TM_MovCmd_ListenNode:='Listen1';
		
			IF (NOT TM_MovCmd_Done) AND (NOT TM_MovCmd_Error) THEN
				Stage:=102;
			END_IF;
		102:
			TM_MovCmd_Execute:=TRUE;
			IF TM_MovCmd_Done THEN;
				Stage:=110;
			ELSIF TM_MovCmd_Error THEN
				Stage:=9999;
			END_IF;
			
			110:
			TM_MovCmd_Enable:=FALSE;
			MovementIndicatorStage:=Stage;
			IF (NOT TM_MovCmd_Done) AND (NOT TM_MovCmd_Error) AND (NOT TM_MovCmd_Busy) THEN
				Stage:=111;
			END_IF;	
		
		111:
			TM_MovCmd_Enable:=TRUE;
			TM_MovCmd_Movement:='Line';
			TM_MovCmd_DataFormat:='CPR';
			TM_MovCmd_Point:=Position5;
			TM_MovCmd_Speed:=50;
			TM_MovCmd_AccelTime:=200;
			TM_MovCmd_Blending:=100;
			TM_MovCmd_PrecisePos:=1;
			TM_MovCmd_RobotPose:='';
			TM_MovCmd_Command:='var_Start_Stitching=20';
			TM_MovCmd_ActivateExit:=TRUE;
			TM_MovCmd_CommandID:=1;
			TM_MovCmd_Execute:=FALSE;
			TM_MovCmd_ListenNode:='Listen1';
		
			IF (NOT TM_MovCmd_Done) AND (NOT TM_MovCmd_Error) THEN
				Stage:=112;
			END_IF;
		112:
			TM_MovCmd_Execute:=TRUE;
			IF TM_MovCmd_Done THEN;
				Stage:=120;
			ELSIF TM_MovCmd_Error THEN
				Stage:=9999;
			END_IF;
			
				
			120:
			TM_MovCmd_Enable:=FALSE;
			MovementIndicatorStage:=Stage;
			IF (NOT TM_MovCmd_Done) AND (NOT TM_MovCmd_Error) AND (NOT TM_MovCmd_Busy) THEN
				Stage:=121;
			END_IF;	
		
		121:
			TM_MovCmd_Enable:=TRUE;
			TM_MovCmd_Movement:='Line';
			TM_MovCmd_DataFormat:='CPR';
			TM_MovCmd_Point:=Position6;
			TM_MovCmd_Speed:=50;
			TM_MovCmd_AccelTime:=200;
			TM_MovCmd_Blending:=100;
			TM_MovCmd_PrecisePos:=1;
			TM_MovCmd_RobotPose:='';
			TM_MovCmd_Command:='var_Start_Stitching=20';
			TM_MovCmd_ActivateExit:=FALSE;
			TM_MovCmd_CommandID:=1;
			TM_MovCmd_Execute:=FALSE;
			TM_MovCmd_ListenNode:='Listen1';
		
			IF (NOT TM_MovCmd_Done) AND (NOT TM_MovCmd_Error) THEN
				Stage:=122;
			END_IF;
		122:
			TM_MovCmd_Execute:=TRUE;
			IF TM_MovCmd_Done THEN;
				Stage:=130;
			ELSIF TM_MovCmd_Error THEN
				Stage:=9999;
			END_IF;
			
			130:
			TM_MovCmd_Enable:=FALSE;
			MovementIndicatorStage:=Stage;
			IF (NOT TM_MovCmd_Done) AND (NOT TM_MovCmd_Error) AND (NOT TM_MovCmd_Busy) THEN
				Stage:=131;
			END_IF;	
		
		131:
			TM_MovCmd_Enable:=TRUE;
			TM_MovCmd_Movement:='Line';
			TM_MovCmd_DataFormat:='CPR';
			TM_MovCmd_Point:=Position7;
			TM_MovCmd_Speed:=50;
			TM_MovCmd_AccelTime:=200;
			TM_MovCmd_Blending:=100;
			TM_MovCmd_PrecisePos:=1;
			TM_MovCmd_RobotPose:='';
			TM_MovCmd_Command:='var_Start_Stitching=20';
			TM_MovCmd_ActivateExit:=FALSE;
			TM_MovCmd_CommandID:=1;
			TM_MovCmd_Execute:=FALSE;
			TM_MovCmd_ListenNode:='Listen1';
		
			IF (NOT TM_MovCmd_Done) AND (NOT TM_MovCmd_Error) THEN
				Stage:=132;
			END_IF;
		132:
			TM_MovCmd_Execute:=TRUE;
			IF TM_MovCmd_Done THEN;
				Stage:=140;
			ELSIF TM_MovCmd_Error THEN
				Stage:=9999;
			END_IF;
			
			140:
			TM_MovCmd_Enable:=FALSE;
			MovementIndicatorStage:=Stage;
			IF (NOT TM_MovCmd_Done) AND (NOT TM_MovCmd_Error) AND (NOT TM_MovCmd_Busy) THEN
				Stage:=141;
			END_IF;	
		
		141:
			TM_MovCmd_Enable:=TRUE;
			TM_MovCmd_Movement:='Line';
			TM_MovCmd_DataFormat:='CPR';
			TM_MovCmd_Point:=Position8;
			TM_MovCmd_Speed:=50;
			TM_MovCmd_AccelTime:=200;
			TM_MovCmd_Blending:=100;
			TM_MovCmd_PrecisePos:=1;
			TM_MovCmd_RobotPose:='';
			TM_MovCmd_Command:='var_Start_Stitching=20';
			TM_MovCmd_ActivateExit:=FALSE;
			TM_MovCmd_CommandID:=1;
			TM_MovCmd_Execute:=FALSE;
			TM_MovCmd_ListenNode:='Listen1';
		
			IF (NOT TM_MovCmd_Done) AND (NOT TM_MovCmd_Error) THEN
				Stage:=142;
			END_IF;
		142:
			TM_MovCmd_Execute:=TRUE;
			IF TM_MovCmd_Done THEN;
				Stage:=150;
			ELSIF TM_MovCmd_Error THEN
				Stage:=9999;
			END_IF;
			
			150:
			TM_MovCmd_Enable:=FALSE;
			MovementIndicatorStage:=Stage;
			IF (NOT TM_MovCmd_Done) AND (NOT TM_MovCmd_Error) AND (NOT TM_MovCmd_Busy) THEN
				Stage:=151;
			END_IF;	
		
		151:
			TM_MovCmd_Enable:=TRUE;
			TM_MovCmd_Movement:='Line';
			TM_MovCmd_DataFormat:='CPR';
			TM_MovCmd_Point:=Position9;
			TM_MovCmd_Speed:=50;
			TM_MovCmd_AccelTime:=200;
			TM_MovCmd_Blending:=100;
			TM_MovCmd_PrecisePos:=1;
			TM_MovCmd_RobotPose:='';
			TM_MovCmd_Command:='var_Start_Stitching=30';
			TM_MovCmd_ActivateExit:=TRUE;
			TM_MovCmd_CommandID:=1;
			TM_MovCmd_Execute:=FALSE;
			TM_MovCmd_ListenNode:='Listen1';
		
			IF (NOT TM_MovCmd_Done) AND (NOT TM_MovCmd_Error) THEN
				Stage:=152;
			END_IF;
		152:
			TM_MovCmd_Execute:=TRUE;
			IF TM_MovCmd_Done THEN;
				Stage:=160;
			ELSIF TM_MovCmd_Error THEN
				Stage:=9999;
			END_IF;
			
			160:
			TM_MovCmd_Enable:=FALSE;
			MovementIndicatorStage:=Stage;
			IF (NOT TM_MovCmd_Done) AND (NOT TM_MovCmd_Error) AND (NOT TM_MovCmd_Busy) THEN
				Stage:=161;
			END_IF;	
		
		161:
			TM_MovCmd_Enable:=TRUE;
			TM_MovCmd_Movement:='Line';
			TM_MovCmd_DataFormat:='CPR';
			TM_MovCmd_Point:=Position10;
			TM_MovCmd_Speed:=50;
			TM_MovCmd_AccelTime:=200;
			TM_MovCmd_Blending:=100;
			TM_MovCmd_PrecisePos:=1;
			TM_MovCmd_RobotPose:='';
			TM_MovCmd_Command:='var_Start_Stitching=30';
			TM_MovCmd_ActivateExit:=FALSE;
			TM_MovCmd_CommandID:=1;
			TM_MovCmd_Execute:=FALSE;
			TM_MovCmd_ListenNode:='Listen1';
		
			IF (NOT TM_MovCmd_Done) AND (NOT TM_MovCmd_Error) THEN
				Stage:=162;
			END_IF;
		162:
			TM_MovCmd_Execute:=TRUE;
			IF TM_MovCmd_Done THEN;
				Stage:=170;
			ELSIF TM_MovCmd_Error THEN
				Stage:=9999;
			END_IF;
			
			170:
			TM_MovCmd_Enable:=FALSE;
			MovementIndicatorStage:=Stage;
			IF (NOT TM_MovCmd_Done) AND (NOT TM_MovCmd_Error) AND (NOT TM_MovCmd_Busy) THEN
				Stage:=171;
			END_IF;	
		
		171:
			TM_MovCmd_Enable:=TRUE;
			TM_MovCmd_Movement:='Line';
			TM_MovCmd_DataFormat:='CPR';
			TM_MovCmd_Point:=Home;
			TM_MovCmd_Speed:=50;
			TM_MovCmd_AccelTime:=200;
			TM_MovCmd_Blending:=100;
			TM_MovCmd_PrecisePos:=1;
			TM_MovCmd_RobotPose:='';
			TM_MovCmd_Command:='var_Start_Stitching=30';
			TM_MovCmd_ActivateExit:=FALSE;
			TM_MovCmd_CommandID:=1;
			TM_MovCmd_Execute:=FALSE;
			TM_MovCmd_ListenNode:='Listen1';
		
			IF (NOT TM_MovCmd_Done) AND (NOT TM_MovCmd_Error) THEN
				Stage:=172;
			END_IF;
		172:
			TM_MovCmd_Execute:=TRUE;
			IF TM_MovCmd_Done THEN;
				Stage:=9999;
			ELSIF TM_MovCmd_Error THEN
				Stage:=9999;
			END_IF;
			
	END_CASE;
	
END_IF;

		//Stitching control based on robot absolute position
		Run_Stiching:=1;
		IF RobotIO.ControlBox.DO0 = 1 AND Stitching_InManual = 0 AND StartProgram = 1 THEN 
				Speed:= 2;
		ELSIF RobotIO.ControlBox.DO0 = 0 AND Stitching_InManual = 0 AND StartProgram = 1 THEN
			Speed:= -2;
		ELSIF RobotIO.ControlBox.DO0 = 0 AND Stitching_InManual = 0 AND Stage = 9999  THEN
			Speed:= 0;
		END_IF;

TM_MovCmd_Instance(
	Done=>TM_MovCmd_Done,
	Busy=>TM_MovCmd_Busy,
	Error=>TM_MovCmd_Error,
	ErrorID=>TM_MovCmd_ErrorID,
	Execute:=TM_MovCmd_Execute,
	RobotID:=ListenNode_Connect_TCP_Socket,
	Movement:=TM_MovCmd_Movement,
	DataFormat:=TM_MovCmd_DataFormat,
	Point:=TM_MovCmd_Point,
	Speed:=TM_MovCmd_Speed,
	AccelTime:=TM_MovCmd_AccelTime,
	Blending:=TM_MovCmd_Blending,
	PrecisePos:=TM_MovCmd_PrecisePos,
	RobotPose:=TM_MovCmd_RobotPose,
	Command:=TM_MovCmd_Command,  
	ActivateExit:=TM_MovCmd_ActivateExit,
	CommandID:=TM_MovCmd_CommandID,
	TimeOut:=T#3600s,
	ListenNode:=TM_MovCmd_ListenNode,
	TimeOutET=>TM_MovCmd_TimeOutET,
	Enable:=TM_MovCmd_Enable
);

TM_ChangeTCP_Instance(
	Enable:=TM_ChangeTCP_Enable,
	Execute:=TM_ChangeTCP_Execute,
	RobotID:=ListenNode_Connect_TCP_Socket,
	TCP:=TM_ChangeTCP_TCP,
	Weight:=TM_ChangeTCP_Weight,
	MomInertia:=TM_ChangeTCP_MomInertia,
	RefFrame:=TM_ChangeTCP_RefFrame,
	Command:=TM_ChangeTCP_Command,
	ActivateExit:=TM_ChangeTCP_ActivateExit,
	ListenNode:=TM_ChangeTCP_ListenNode,
	TimeOut:=T#3600s,
	CommandID:=TM_ChangeTCP_CommandID,
	Done=>TM_ChangeTCP_Done,
	Busy=>TM_ChangeTCP_Busy,
	Error=>TM_ChangeTCP_Error,
	ErrorID=>TM_ChangeTCP_ErrorID,
	TimeOutET=>TM_ChangeTCP_TimeOutET
);

TM_ChangeLoad_Instance(
	Enable:=TM_ChangeLoad_Enable,
	Execute:=TM_ChangeLoad_Execute,
	RobotID:=ListenNode_Connect_TCP_Socket,
	Payload:=TM_ChangeLoad_Payload,
	Command:=TM_ChangeLoad_Command,
	ActivateExit:=TM_ChangeLoad_ActivateExit,
	ListenNode:=TM_ChangeLoad_ListenNode,
	TimeOut:=T#3600s,
	CommandID:=TM_ChangeLoad_CommandID,
	Done=>TM_ChangeLoad_Done,
	Busy=>TM_ChangeLoad_Busy,
	Error=>TM_ChangeLoad_Error,
	ErrorID=>TM_ChangeLoad_ErrorID,
	TimeOutET=>TM_ChangeLoad_TimeOutET
);

TM_CircleCmd_Instance(
	Enable:=TM_CircleCmd_Enable,
	Execute:=TM_CircleCmd_Execute,
	RobotID:=ListenNode_Connect_TCP_Socket,
	DataFormat:=TM_CircleCmd_DataFormat,
	ArcPoint:=TM_CircleCmd_ArcPoint,
	EndArcPoint:=TM_CircleCmd_EndArcPoint,
	Speed:=TM_CircleCmd_Speed,
	AccelTime:=TM_CircleCmd_AccelTime,
	Blending:=TM_CircleCmd_Blending,
	ArcAngle:=TM_CircleCmd_ArcAngle,
	PrecisePos:=TM_CircleCmd_PrecisePos,
	Command:=TM_CircleCmd_Command,
	ActivateExit:=TM_CircleCmd_ActivateExit,
	ListenNode:=TM_CircleCmd_ListenNode,
	TimeOut:=T#3600s,
	CommandID:=TM_CircleCmd_CommandID,
	Done=>TM_CircleCmd_Done,
	Busy=>TM_CircleCmd_Busy,
	Error=>TM_CircleCmd_Error,
	ErrorID=>TM_CircleCmd_ErrorID,
	TimeOutET=>TM_CircleCmd_TimeOutET
);

TM_ChangeBase_Instance(
	Enable:=TM_ChangeBase_Enable,
	Execute:=TM_ChangeBase_Execute,
	RobotID:=ListenNode_Connect_TCP_Socket,
	Base:=TM_ChangeBase_Base,
	Command:=TM_ChangeBase_Command,
	ActivateExit:=TM_ChangeBase_ActivateExit,
	ListenNode:=TM_ChangeBase_ListenNode,
	TimeOut:=T#3600s,
	CommandID:=TM_ChangeBase_CommandID,
	Done=>TM_ChangeBase_Done,
	Busy=>TM_ChangeBase_Busy,
	Error=>TM_ChangeBase_Error,
	ErrorID=>TM_ChangeBase_ErrorID,
	TimeOutET=>TM_ChangeBase_TimeOutET
);
END_PROGRAM

PROGRAM CobotModbusComms
VAR
    ButtonStatus : TMmodbus\sRobotStickButtons;
    TM_Modbus : TMmodbus\fbTMmodbus1_80;
    PortIsReady : BOOL;
END_VAR
VAR_EXTERNAL
    StartCommunications : BOOL;
    MBerror : WORD;
    RobotCoordinates : TMmodbus\sRobotCoordinate;  (* Standard robot coordinates *)
    TouchCoordinates : TMmodbus\sRobotCoordinateTouch;  (* Robot coordinates coming from the 'Touch Stop' node. *)
    RobotStatus : TMmodbus\sRobotStatus;
    RobotVitals : TMmodbus\sRobotVitals;
    Config : TMmodbus\sConfiguration;
    RobotTCPLive : TMmodbus\sRobotTCPLive;
    CurrentProjectName : string[200];
    NewProjectName : string[200];
    CommsRoundRobin : REAL;
    TCPerror : WORD;
    RobotControlBoxInfo : TMmodbus\sRobotControllerData;
    Buttons : TMmodbus\sRobotStickButtons;
    RobotIO : TMmodbus\sRobotIO;
    RobotSafetySettings : TMmodbus\sRobotSafety;
    RealsToRobot : ARRAY[0..49] OF real;
    FloatsFromRobot : ARRAY[0..49] OF real;
    BoolsToRobot : ARRAY[0..63] OF BOOL;
    Int16sFromRobot : ARRAY[0..49] OF INT;
    BoolsFromRobot : ARRAY[0..63] OF BOOL;
    IntsToRobot : ARRAY[0..49] OF INT;
    CommunicationsStatus : _eCONNECTION_STATE;
    CommunicationsBusy : BOOL;
    RetryCounter : UINT;
    TCPerrorOriginator : TMModbus\eFunctionBlockError;
    RobotJointTorques : TMmodbus\sRobotJointTorque;
    TaskTimeFB : REAL;
END_VAR
VAR
    _e1 : R_TRIG;
    _e2 : F_TRIG;
END_VAR

(* Section TM12ModbusComms: ladder, written here as Structured Text *)

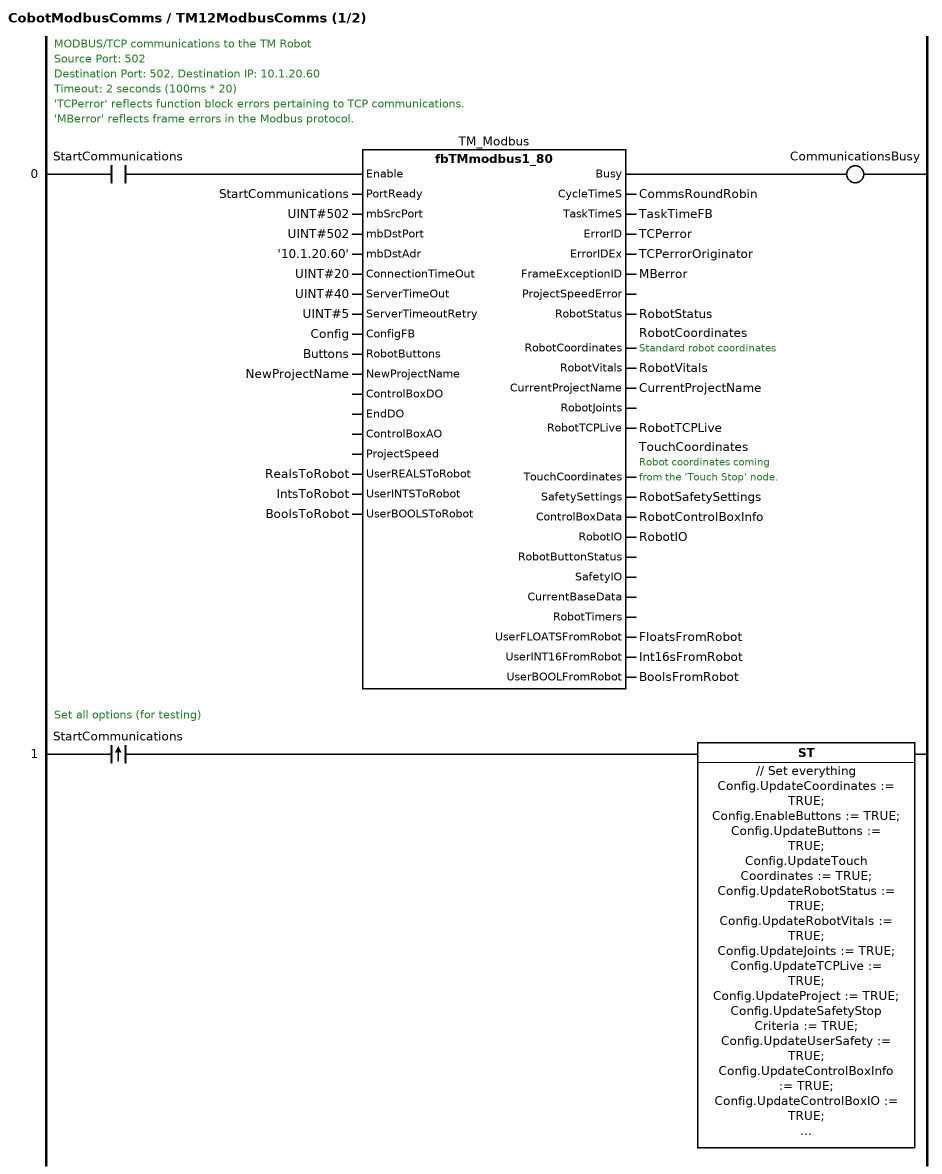
(* Rung 0: MODBUS/TCP communications to the TM Robot / Source Port: 502 / Destination Port: 502, Destination IP: 10.1.20.60 / Timeout: 2 seconds (100ms * 20) / 'TCPerror' reflects function block errors pertaining to TCP communications. / 'MBerror' reflects frame errors in the Modbus protocol. *)
TM_Modbus(Enable := StartCommunications, PortReady := StartCommunications, mbSrcPort := UINT#502, mbDstPort := UINT#502, mbDstAdr := '10.1.20.60', ConnectionTimeOut := UINT#20, ServerTimeOut := UINT#40, ServerTimeoutRetry := UINT#5, ConfigFB := Config, RobotButtons := Buttons, NewProjectName := NewProjectName, UserREALSToRobot := RealsToRobot, UserINTSToRobot := IntsToRobot, UserBOOLSToRobot := BoolsToRobot, CycleTimeS => CommsRoundRobin, TaskTimeS => TaskTimeFB, ErrorID => TCPerror, ErrorIDEx => TCPerrorOriginator, FrameExceptionID => MBerror, RobotStatus => RobotStatus, RobotCoordinates => RobotCoordinates, RobotVitals => RobotVitals, CurrentProjectName => CurrentProjectName, RobotTCPLive => RobotTCPLive, TouchCoordinates => TouchCoordinates, SafetySettings => RobotSafetySettings, ControlBoxData => RobotControlBoxInfo, RobotIO => RobotIO, UserFLOATSFromRobot => FloatsFromRobot, UserINT16FromRobot => Int16sFromRobot, UserBOOLFromRobot => BoolsFromRobot);
CommunicationsBusy := TM_Modbus.Busy;
(* Rung 1: Set all options (for testing) *)
_e1(CLK := StartCommunications);
IF _e1.Q THEN
    // Set everything
    Config.UpdateCoordinates := TRUE;
    Config.EnableButtons := TRUE;
    Config.UpdateButtons := TRUE;
    Config.UpdateTouchCoordinates := TRUE;
    Config.UpdateRobotStatus := TRUE;
    Config.UpdateRobotVitals := TRUE;
    Config.UpdateJoints := TRUE;
    Config.UpdateTCPLive := TRUE;
    Config.UpdateProject := TRUE;
    Config.UpdateSafetyStopCriteria := TRUE;
    Config.UpdateUserSafety := TRUE;
    Config.UpdateControlBoxInfo := TRUE;
    Config.UpdateControlBoxIO := TRUE;
    Config.UpdateEndIO := TRUE;
    Config.UpdateSafetyIO := TRUE;
    Config.UpdateUserFLOATS := TRUE;
    Config.UpdateUserINT16 := TRUE;
    Config.UpdateUserCoils := TRUE;
    Config.EnableControlBoxDO := TRUE;
    Config.EnableControlBoxAO := TRUE;
    Config.EnableEndEffectorDO := TRUE;
    Config.UpdateBase := TRUE;
    Config.UpdateTimers := TRUE;
    Config.EnableSpeedChange := TRUE;
END_IF;

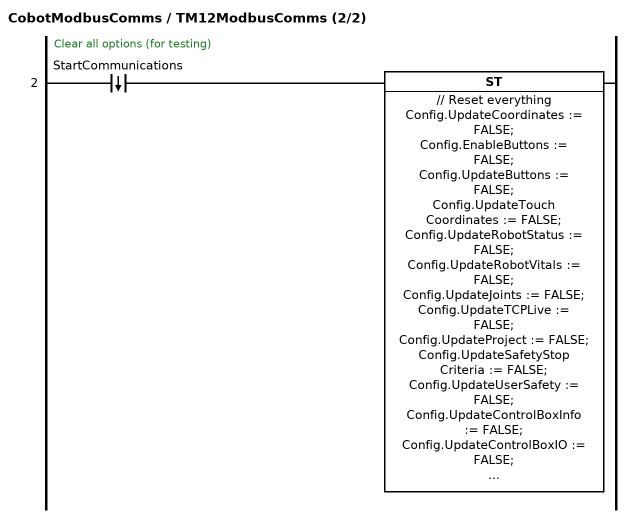
(* Rung 2: Clear all options (for testing) *)
_e2(CLK := StartCommunications);
IF _e2.Q THEN
    // Reset everything
    Config.UpdateCoordinates := FALSE;
    Config.EnableButtons := FALSE;
    Config.UpdateButtons := FALSE;
    Config.UpdateTouchCoordinates := FALSE;
    Config.UpdateRobotStatus := FALSE;
    Config.UpdateRobotVitals := FALSE;
    Config.UpdateJoints := FALSE;
    Config.UpdateTCPLive := FALSE;
    Config.UpdateProject := FALSE;
    Config.UpdateSafetyStopCriteria := FALSE;
    Config.UpdateUserSafety := FALSE;
    Config.UpdateControlBoxInfo := FALSE;
    Config.UpdateControlBoxIO := FALSE;
    Config.UpdateEndIO := FALSE;
    Config.UpdateSafetyIO := FALSE;
    Config.UpdateUserFLOATS := FALSE;
    Config.UpdateUserINT16 := FALSE;
    Config.UpdateUserCoils := FALSE;
    Config.EnableControlBoxDO := FALSE;
    Config.EnableControlBoxAO := FALSE;
    Config.EnableEndEffectorDO := FALSE;
    Config.UpdateBase := FALSE;
    Config.UpdateTimers := FALSE;
    Config.EnableSpeedChange := FALSE;
END_IF;
END_PROGRAM